INTERFACE PUBLIC I_StartingCommands

METHOD PUBLIC Abort
END_METHOD

METHOD PUBLIC StateComplete
END_METHOD

END_INTERFACE

(* stored: Version 1.1.0.1, ProductVersion 3.1.4026.6
   Itf I_StartingCommands: Id {dbee54f7-1ba1-0294-0b8c-497189d1fd31}
   Method Abort: Id {c79c1a54-d781-4585-a291-0aef57d2344b}
   Method StateComplete: Id {b2cdb4af-05c0-47c8-a414-af6e38aeb8b7} *)
